TYPE ST_ClampStationParCfg :
STRUCT
    SchemaVersion : UINT := 1;
END_STRUCT
END_TYPE

(* stored: Version 1.1.0.1, ProductVersion 3.1.4024.12
   DUT ST_ClampStationParCfg: Id {54d45e6f-83f3-4ce7-9b51-779353720187} *)
